TYPE ES_M :
STRUCT
END_STRUCT
END_TYPE

(* stored: Version 1.1.0.1, ProductVersion 3.1.4022.6
   DUT ES_M: Id {656eb773-c3b4-4739-8c1d-cca043e06e39} *)
